TYPE ST_StopParams :
STRUCT
	Deceleration	: LREAL;
	Jerk			: LREAL;
END_STRUCT
END_TYPE

(* stored: Version 1.1.0.1, ProductVersion 3.1.4023.8
   DUT ST_StopParams: Id {2b5884c2-071d-4455-a635-d9a89defea78} *)
